{attribute 'qualified_only'}
VAR_GLOBAL

    // Par
    {attribute 'OPC.UA.DA' := '1'}
    {attribute 'OPC.UA.DA.StructuredType' := '1'}
    g_stBigBagDischargePar        : ST_BigBagDischargePar;

    // Status
    {attribute 'OPC.UA.DA' := '1'}
    {attribute 'OPC.UA.DA.StructuredType' := '1'}
    g_stBigBagDischargeStatus     : ST_BigBagDischargeStatus;

    // OutValues
    {attribute 'OPC.UA.DA' := '1'}
    {attribute 'OPC.UA.DA.StructuredType' := '1'}
    g_stBigBagDischargeOutValues  : ST_BigBagDischargeOutValues;

END_VAR

(* stored: Version 1.1.0.1, ProductVersion 3.1.4024.16
   GVL GVL_BigBagDischarge: Id {67dff12f-69c0-4986-8d48-09df0faf3ac7} *)
